{attribute 'OPC.UA.DA' := '1'}
FUNCTION_BLOCK FB_TwoPosActuator
VAR_INPUT
    {attribute 'OPC.UA.DA' := '0'}
    EnableIn : BOOL := TRUE;
    
    // Permissive inputs (INT with -1 = all OK)
    {attribute 'OPC.UA.DA' := '0'}
    inPermAdv : INT := -1;
    {attribute 'OPC.UA.DA' := '0'}
    inPermRet : INT := -1;
    
    // Configuration
    {attribute 'OPC.UA.DA' := '1'}
    {attribute 'OPC.UA.DA.Access' := '1'}
    cfg : ST_TwoPosActuator_Cfg;
END_VAR

VAR_OUTPUT
    {attribute 'OPC.UA.DA' := '0'}
    EnableOut : BOOL;
    {attribute 'OPC.UA.DA' := '1'}
    {attribute 'OPC.UA.DA.Access' := '1'}
    sts : ST_TwoPosActuator_Sts;
END_VAR

VAR_IN_OUT
    {attribute 'OPC.UA.DA' := '0'}
    IO : ST_TwoPosActuator_IO;
END_VAR

VAR
    // Composed modules - permissive handlers (visible on OPC)
    advancePermissives : FB_Permissives;
    retractPermissives : FB_Permissives;
    
    // Internal state machine
    {attribute 'OPC.UA.DA' := '0'}
    currentState : E_TwoPosActuator_State := E_TwoPosActuator_State.Undefined;
    {attribute 'OPC.UA.DA' := '0'}
    previousState : E_TwoPosActuator_State;
    
    // Timers for motion
    {attribute 'OPC.UA.DA' := '0'}
    advanceTimer : TON;
    {attribute 'OPC.UA.DA' := '0'}
    retractTimer : TON;
    
    // Edge detection
    {attribute 'OPC.UA.DA' := '0'}
    rTrigAdvanced : R_TRIG;
    {attribute 'OPC.UA.DA' := '0'}
    rTrigRetracted : R_TRIG;
    
    // Internal flags
    {attribute 'OPC.UA.DA' := '0'}
    bothFeedbackActive : BOOL;
    
    // Fault handling
    {attribute 'OPC.UA.DA' := '0'}
    faultLatched : BOOL;
    {attribute 'OPC.UA.DA' := '0'}
    lastFault : E_TwoPosActuator_Fault;
    {attribute 'OPC.UA.DA' := '0'}
    permIdx : INT;
    
    // Source control
    {attribute 'OPC.UA.DA' := '0'}
    bSourceLockedToProg : BOOL;
END_VAR

//-----------------------------------------------------------------------------
// Main Implementation - FB_TwoPosActuator
// Cyclic monitoring only. All commands issued via methods.
//-----------------------------------------------------------------------------
EnableOut := EnableIn;

IF EnableIn THEN
    
    //-------------------------------------------------------------------------
    // Permissive Evaluation
    //-------------------------------------------------------------------------
    FOR permIdx := 0 TO 15 DO
        advancePermissives.MapReason(
            nIndex := permIdx,
            sDescription := advancePermissives.cfg.Desc[permIdx],
            bValue := (inPermAdv AND SHL(1, permIdx)) <> 0
        );
    END_FOR;
    advancePermissives();
    
    FOR permIdx := 0 TO 15 DO
        retractPermissives.MapReason(
            nIndex := permIdx,
            sDescription := retractPermissives.cfg.Desc[permIdx],
            bValue := (inPermRet AND SHL(1, permIdx)) <> 0
        );
    END_FOR;
    retractPermissives();
    
    //-------------------------------------------------------------------------
    // Feedback Analysis
    //-------------------------------------------------------------------------
    bothFeedbackActive := IO.inFbkAdvanced AND IO.inFbkRetracted;
    
    //-------------------------------------------------------------------------
    // State Machine - Cyclic Monitoring
    // Methods set currentState and IO; body monitors for completion/faults.
    //-------------------------------------------------------------------------
    previousState := currentState;
    
    CASE currentState OF
        
        E_TwoPosActuator_State.Undefined:
            IO.outValveAdvance := FALSE;
            IO.outValveRetract := FALSE;
            
            IF bothFeedbackActive THEN
                currentState := E_TwoPosActuator_State.Fault;
                sts.faultCode := E_TwoPosActuator_Fault.BothFeedbackOn;
                faultLatched := TRUE;
            ELSIF IO.inFbkAdvanced AND NOT IO.inFbkRetracted THEN
                currentState := E_TwoPosActuator_State.Advanced;
            ELSIF IO.inFbkRetracted AND NOT IO.inFbkAdvanced THEN
                currentState := E_TwoPosActuator_State.Retracted;
            END_IF;
        
        E_TwoPosActuator_State.Retracted:
            IF cfg.cfgHoldAtRetracted THEN
                IO.outValveRetract := TRUE;
            ELSE
                IO.outValveRetract := FALSE;
            END_IF;
            IO.outValveAdvance := FALSE;
            
            IF bothFeedbackActive THEN
                currentState := E_TwoPosActuator_State.Fault;
                sts.faultCode := E_TwoPosActuator_Fault.BothFeedbackOn;
                faultLatched := TRUE;
            ELSIF NOT IO.inFbkRetracted THEN
                currentState := E_TwoPosActuator_State.Fault;
                sts.faultCode := E_TwoPosActuator_Fault.UndefinedState;
                faultLatched := TRUE;
            END_IF;
        
        E_TwoPosActuator_State.Advancing:
            IO.outValveAdvance := TRUE;
            IO.outValveRetract := FALSE;
            advanceTimer(IN := TRUE, PT := DINT_TO_TIME(cfg.cfgAdvTimeoutS * 1000));
            
            IF IO.inFbkAdvanced AND NOT IO.inFbkRetracted THEN
                currentState := E_TwoPosActuator_State.Advanced;
                advanceTimer(IN := FALSE);
            ELSIF advanceTimer.Q THEN
                currentState := E_TwoPosActuator_State.Fault;
                sts.faultCode := E_TwoPosActuator_Fault.AdvanceTimeout;
                faultLatched := TRUE;
                advanceTimer(IN := FALSE);
            ELSIF bothFeedbackActive THEN
                currentState := E_TwoPosActuator_State.Fault;
                sts.faultCode := E_TwoPosActuator_Fault.BothFeedbackOn;
                faultLatched := TRUE;
                advanceTimer(IN := FALSE);
            ELSIF NOT advancePermissives.sts.OK THEN
                currentState := E_TwoPosActuator_State.Fault;
                sts.faultCode := E_TwoPosActuator_Fault.PermissivesNotOK;
                faultLatched := TRUE;
                advanceTimer(IN := FALSE);
            END_IF;
        
        E_TwoPosActuator_State.Advanced:
            IF cfg.cfgHoldAtAdvanced THEN
                IO.outValveAdvance := TRUE;
            ELSE
                IO.outValveAdvance := FALSE;
            END_IF;
            IO.outValveRetract := FALSE;
            
            IF bothFeedbackActive THEN
                currentState := E_TwoPosActuator_State.Fault;
                sts.faultCode := E_TwoPosActuator_Fault.BothFeedbackOn;
                faultLatched := TRUE;
            ELSIF NOT IO.inFbkAdvanced THEN
                currentState := E_TwoPosActuator_State.Fault;
                sts.faultCode := E_TwoPosActuator_Fault.UndefinedState;
                faultLatched := TRUE;
            END_IF;
        
        E_TwoPosActuator_State.Retracting:
            IO.outValveRetract := TRUE;
            IO.outValveAdvance := FALSE;
            retractTimer(IN := TRUE, PT := DINT_TO_TIME(cfg.cfgRetTimeoutS * 1000));
            
            IF IO.inFbkRetracted AND NOT IO.inFbkAdvanced THEN
                currentState := E_TwoPosActuator_State.Retracted;
                retractTimer(IN := FALSE);
            ELSIF retractTimer.Q THEN
                currentState := E_TwoPosActuator_State.Fault;
                sts.faultCode := E_TwoPosActuator_Fault.RetractTimeout;
                faultLatched := TRUE;
                retractTimer(IN := FALSE);
            ELSIF bothFeedbackActive THEN
                currentState := E_TwoPosActuator_State.Fault;
                sts.faultCode := E_TwoPosActuator_Fault.BothFeedbackOn;
                faultLatched := TRUE;
                retractTimer(IN := FALSE);
            ELSIF NOT retractPermissives.sts.OK THEN
                currentState := E_TwoPosActuator_State.Fault;
                sts.faultCode := E_TwoPosActuator_Fault.PermissivesNotOK;
                faultLatched := TRUE;
                retractTimer(IN := FALSE);
            END_IF;
        
        E_TwoPosActuator_State.Fault:
            IO.outValveAdvance := FALSE;
            IO.outValveRetract := FALSE;
            advanceTimer(IN := FALSE);
            retractTimer(IN := FALSE);
    END_CASE;
    
    //-------------------------------------------------------------------------
    // Status Output Generation
    //-------------------------------------------------------------------------
    sts.state := currentState;
    sts.stsAdvanced := (currentState = E_TwoPosActuator_State.Advanced);
    sts.stsRetracted := (currentState = E_TwoPosActuator_State.Retracted);
    sts.stsMoving := (currentState = E_TwoPosActuator_State.Advancing) OR 
                     (currentState = E_TwoPosActuator_State.Retracting);
    sts.stsFaulted := (currentState = E_TwoPosActuator_State.Fault) OR faultLatched;
    sts.lastFaultCode := lastFault;
    
    rTrigAdvanced(CLK := sts.stsAdvanced);
    sts.osAdvanced := rTrigAdvanced.Q;
    
    rTrigRetracted(CLK := sts.stsRetracted);
    sts.osRetracted := rTrigRetracted.Q;
    
    //-------------------------------------------------------------------------
    // String Generation for OPC/HMI
    //-------------------------------------------------------------------------
    CASE currentState OF
        E_TwoPosActuator_State.Undefined:   sts.stateString := 'Undefined';
        E_TwoPosActuator_State.Retracted:   sts.stateString := 'Retracted';
        E_TwoPosActuator_State.Advancing:   sts.stateString := 'Advancing';
        E_TwoPosActuator_State.Advanced:    sts.stateString := 'Advanced';
        E_TwoPosActuator_State.Retracting:  sts.stateString := 'Retracting';
        E_TwoPosActuator_State.Fault:       sts.stateString := 'Fault';
    ELSE
        sts.stateString := 'Unknown';
    END_CASE;
    
    CASE sts.faultCode OF
        E_TwoPosActuator_Fault.None:               sts.faultString := 'No Fault';
        E_TwoPosActuator_Fault.AdvanceTimeout:      sts.faultString := 'Advance Timeout';
        E_TwoPosActuator_Fault.RetractTimeout:      sts.faultString := 'Retract Timeout';
        E_TwoPosActuator_Fault.BothFeedbackOn:      sts.faultString := 'Both Feedbacks Active';
        E_TwoPosActuator_Fault.UndefinedState:      sts.faultString := 'Position Undefined';
        E_TwoPosActuator_Fault.PermissivesNotOK:    sts.faultString := 'Permissives Not OK';
        E_TwoPosActuator_Fault.ConflictingCommands:  sts.faultString := 'Conflicting Commands';
        E_TwoPosActuator_Fault.NoFeedback:          sts.faultString := 'No Position Feedback';
    ELSE
        sts.faultString := 'Unknown Fault';
    END_CASE;
    
    CASE sts.lastFaultCode OF
        E_TwoPosActuator_Fault.None:               sts.lastFaultString := 'No Previous Fault';
        E_TwoPosActuator_Fault.AdvanceTimeout:      sts.lastFaultString := 'Last: Advance Timeout';
        E_TwoPosActuator_Fault.RetractTimeout:      sts.lastFaultString := 'Last: Retract Timeout';
        E_TwoPosActuator_Fault.BothFeedbackOn:      sts.lastFaultString := 'Last: Both Feedbacks Active';
        E_TwoPosActuator_Fault.UndefinedState:      sts.lastFaultString := 'Last: Position Undefined';
        E_TwoPosActuator_Fault.PermissivesNotOK:    sts.lastFaultString := 'Last: Permissives Not OK';
        E_TwoPosActuator_Fault.ConflictingCommands:  sts.lastFaultString := 'Last: Conflicting Commands';
        E_TwoPosActuator_Fault.NoFeedback:          sts.lastFaultString := 'Last: No Position Feedback';
    ELSE
        sts.lastFaultString := 'Last: Unknown Fault';
    END_CASE;
    
ELSE
    IO.outValveAdvance := FALSE;
    IO.outValveRetract := FALSE;
    advanceTimer(IN := FALSE);
    retractTimer(IN := FALSE);
END_IF;

{attribute 'TcRpcEnable' := '1'}
METHOD PUBLIC Advance : E_RpcMethodResponse
VAR_INPUT
    eRequester : E_Requester := E_Requester.PROG;
END_VAR
// 1. Source + fault validation
Advance := F_ValidateRequester(eRequester, bSourceLockedToProg, faultLatched, FALSE, FALSE);
IF Advance <> E_RpcMethodResponse.ACCEPTED THEN RETURN; END_IF;

// 2. State check — must not already be advanced or advancing
IF currentState = E_TwoPosActuator_State.Advanced OR currentState = E_TwoPosActuator_State.Advancing THEN
    Advance := E_RpcMethodResponse.REJECTED_ALREADY_AT_TARGET;
    RETURN;
END_IF;

// 3. Permissive check
IF NOT advancePermissives.sts.OK THEN
    Advance := E_RpcMethodResponse.REJECTED_PERMISSIVE_NOT_MET;
    RETURN;
END_IF;

// 4. Execute — set state, body handles the rest
currentState := E_TwoPosActuator_State.Advancing;
advanceTimer(IN := FALSE);
Advance := E_RpcMethodResponse.ACCEPTED;
END_METHOD

{attribute 'TcRpcEnable' := '1'}
METHOD PUBLIC Retract : E_RpcMethodResponse
VAR_INPUT
    eRequester : E_Requester := E_Requester.PROG;
END_VAR
// 1. Source + fault validation
Retract := F_ValidateRequester(eRequester, bSourceLockedToProg, faultLatched, FALSE, FALSE);
IF Retract <> E_RpcMethodResponse.ACCEPTED THEN RETURN; END_IF;

// 2. State check — must not already be retracted or retracting
IF currentState = E_TwoPosActuator_State.Retracted OR currentState = E_TwoPosActuator_State.Retracting THEN
    Retract := E_RpcMethodResponse.REJECTED_ALREADY_AT_TARGET;
    RETURN;
END_IF;

// 3. Permissive check
IF NOT retractPermissives.sts.OK THEN
    Retract := E_RpcMethodResponse.REJECTED_PERMISSIVE_NOT_MET;
    RETURN;
END_IF;

// 4. Execute — set state, body handles the rest
currentState := E_TwoPosActuator_State.Retracting;
retractTimer(IN := FALSE);
Retract := E_RpcMethodResponse.ACCEPTED;
END_METHOD

{attribute 'TcRpcEnable' := '1'}
METHOD PUBLIC AllOff : E_RpcMethodResponse
VAR_INPUT
    eRequester : E_Requester := E_Requester.PROG;
END_VAR
// AllOff is always accepted — safety command
AllOff := F_ValidateRequester(eRequester, bSourceLockedToProg, faultLatched, FALSE, TRUE);
IF AllOff <> E_RpcMethodResponse.ACCEPTED THEN RETURN; END_IF;

IO.outValveAdvance := FALSE;
IO.outValveRetract := FALSE;
advanceTimer(IN := FALSE);
retractTimer(IN := FALSE);
currentState := E_TwoPosActuator_State.Undefined;
AllOff := E_RpcMethodResponse.ACCEPTED;
END_METHOD

{attribute 'TcRpcEnable' := '1'}
METHOD PUBLIC Reset : E_RpcMethodResponse
VAR_INPUT
    eRequester : E_Requester := E_Requester.PROG;
END_VAR
// 1. Source validation — allow when faulted
Reset := F_ValidateRequester(eRequester, bSourceLockedToProg, faultLatched, TRUE, FALSE);
IF Reset <> E_RpcMethodResponse.ACCEPTED THEN RETURN; END_IF;

// 2. Must be in fault state
IF currentState <> E_TwoPosActuator_State.Fault THEN
    Reset := E_RpcMethodResponse.REJECTED_WRONG_STATE;
    RETURN;
END_IF;

// 3. Execute — clear fault and go to Undefined for re-evaluation
lastFault := sts.faultCode;
faultLatched := FALSE;
sts.faultCode := E_TwoPosActuator_Fault.None;
currentState := E_TwoPosActuator_State.Undefined;
IO.outValveAdvance := FALSE;
IO.outValveRetract := FALSE;
Reset := E_RpcMethodResponse.ACCEPTED;
END_METHOD

{attribute 'TcRpcEnable' := '1'}
METHOD PUBLIC LockSource : E_RpcMethodResponse
VAR_INPUT
    bLock : BOOL;
END_VAR
bSourceLockedToProg := bLock;
LockSource := E_RpcMethodResponse.ACCEPTED;
END_METHOD

END_FUNCTION_BLOCK

(* stored: Version 1.1.0.1, ProductVersion 3.1.4026.12
   POU FB_TwoPosActuator: Id {a1234567-1234-1234-1234-123456789007}, SpecialFunc None
   Method Advance: Id {a1234567-1234-1234-1234-12345678A001}
   Method Retract: Id {a1234567-1234-1234-1234-12345678A002}
   Method AllOff: Id {a1234567-1234-1234-1234-12345678A003}
   Method Reset: Id {a1234567-1234-1234-1234-12345678A004}
   Method LockSource: Id {a1234567-1234-1234-1234-12345678A005} *)
